(* Logix 5000 project; controller HP_SSC01hv vendor 1 type 14 code 158 rev 32.11; software revision 32.03; part 3 of 15 *)
(* tags used below, declared in another part *)
   A_C1_0218 : ALIAS FOR S_C1_FaultSafety.18;
   A_C1_0219 : ALIAS FOR S_C1_FaultSafety.19;
   A_C1_0220 : ALIAS FOR S_C1_FaultSafety.20;
   A_C1_0221 : ALIAS FOR S_C1_FaultSafety.21;
   A_C1_0222 : ALIAS FOR S_C1_FaultSafety.22;
   A_C1_0223 : ALIAS FOR S_C1_FaultSafety.23;
   A_C1_0311 : ALIAS FOR C1_FaultStandard.11;
   A_C1_0312 : ALIAS FOR C1_FaultStandard.12;
   A_C1_0313 : ALIAS FOR C1_FaultStandard.13;
   A_C1_0314 : ALIAS FOR C1_FaultStandard.14;
   A_C1_0315 : ALIAS FOR C1_FaultStandard.15;
   C1_EncoderDegree : REAL;
   C1_EncoderPositionAtHome : DINT;
   C1_ExcecutePBHoldTimer : TIMER;
   C1_FaultHomeSwitchNotFound : BOOL;
   C1_Homed : BOOL;
   C1_HomeDelay : TIMER[16];
   C1_HomeFindSwitchMAM01 : MOTION_INSTRUCTION;
   C1_HomeFindSwitchMAM02 : MOTION_INSTRUCTION;
   C1_HomeFindSwitchMAS01 : MOTION_INSTRUCTION;
   C1_HomeGetCloseToSwitchMAM01 : MOTION_INSTRUCTION;
   C1_HomeGoToOnPathMAM01 : MOTION_INSTRUCTION;
   C1_HomeMessageNumber : DINT;
   C1_HomeSensorTestMAM02 : MOTION_INSTRUCTION;
   C1_HomeSequence : DINT;
   C1_HomeSequenceAlarms : DINT;
   C1_HomeSequenceAlarmTimer : TIMER[32];
   C1_HomeSequenceInProcess : BOOL;
   C1_HomeSequenceMAH : MOTION_INSTRUCTION;
   C1_HomeSwitchFaultK7KFailedOff : BOOL;
   C1_HomeSwitchFaultK7KFailedOn : BOOL;
   C1_HomeSwitchFaultSafeFailedOff : BOOL;
   C1_HomeSwitchFaultSafeFailedOn : BOOL;
   C1_HomeTest : REAL;
   C1_IndexEnable : BOOL;
   C1_IndexEnableTOF : TIMER;
   C1_IndexMAM01 : MOTION_INSTRUCTION;
   C1_IndexMAS01 : MOTION_INSTRUCTION;
   C1_IndexMessageNumber : DINT;
   C1_IndexPermissive : BOOL;
   C1_Jog_ONS : DINT;
   C1_JogDirection : DINT;
   C1_JogEnable : BOOL;
   C1_JogEnableTOF : TIMER;
   C1_JogForwardFastSelected : BOOL;
   C1_JogForwardSlowSelected : BOOL;
   C1_JogMAJ01 : MOTION_INSTRUCTION;
   C1_JogMAJ02 : MOTION_INSTRUCTION;
   C1_JogMAS01 : MOTION_INSTRUCTION;
   C1_JogMessageNumber : DINT;
   C1_JogPermissive : BOOL;
   C1_JogReverseFastSelected : BOOL;
   C1_JogReverseSlowSelected : BOOL;
   C1_MAJAcceleration : REAL;
   C1_MAJDeceleration : REAL;
   C1_MAJSpeed : REAL;
   C1_OIT_Current : DINT;
   C1_RemoteHomeCMD : BOOL;
   C1_ServoActionStatusOnDelay : TIMER;
   C1_SetEncoderHomePosition : BOOL;
   C1HomeSensorTestMAM01 : MOTION_INSTRUCTION;
   C1HomeSequenceONS : BOOL;
   C1HomeSequenceONS2 : BOOL;
   none : BOOL;
   S_C1_EncoderPositionAtHomeSet : BOOL;
   S_C1_ExecutePB : BOOL;
   S_C1_FaultReset : BOOL;
   S_C1_HomeSafePE : ALIAS FOR C1_Safe:I.Pt04Data;
   S_C1_ModeLocal : BOOL;
   S_C1_ModeRemote : BOOL;
   S_C1_MSTOP_InputOK : BOOL;
   S_EncoderCtsFor360Deg : DINT;
(* Carousel1, continued *)

ROUTINE C130_Home   (* ladder *)
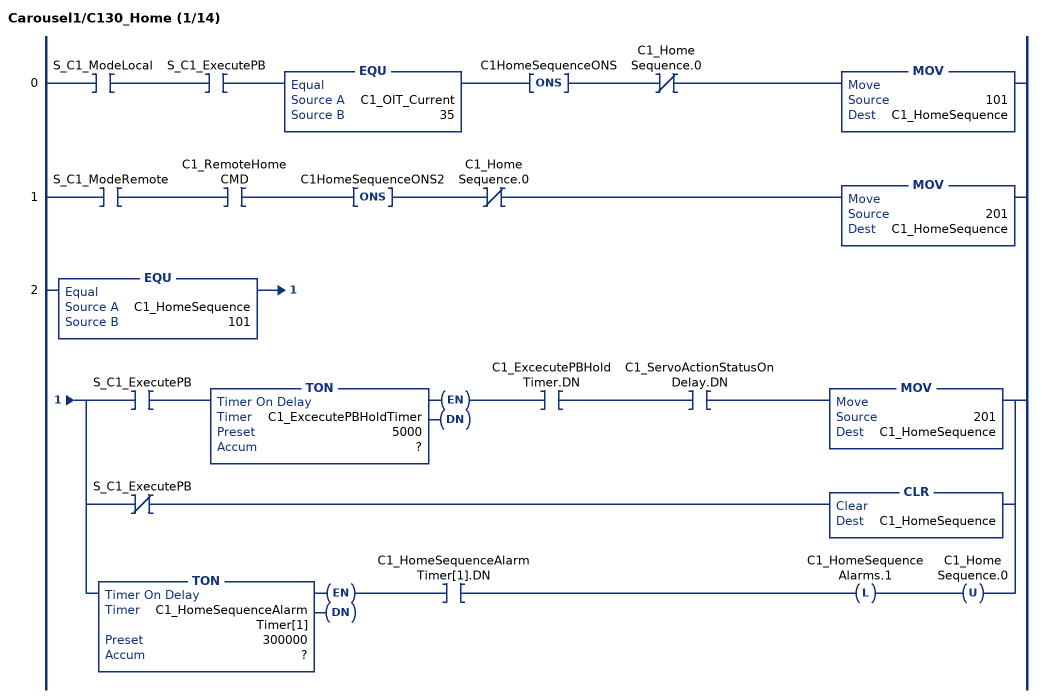
   0: XIC(S_C1_ModeLocal)XIC(S_C1_ExecutePB)EQU(C1_OIT_Current,35)ONS(C1HomeSequenceONS)XIO(C1_HomeSequence.0)MOV(101,C1_HomeSequence);
   1: XIC(S_C1_ModeRemote)XIC(C1_RemoteHomeCMD)ONS(C1HomeSequenceONS2)XIO(C1_HomeSequence.0)MOV(201,C1_HomeSequence);
   2: EQU(C1_HomeSequence,101)[XIC(S_C1_ExecutePB) TON(C1_ExcecutePBHoldTimer,?,?) XIC(C1_ExcecutePBHoldTimer.DN) XIC(C1_ServoActionStatusOnDelay.DN) MOV(201,C1_HomeSequence) ,XIO(S_C1_ExecutePB) CLR(C1_HomeSequence) ,TON(C1_HomeSequenceAlarmTimer[1],?,?) XIC(C1_HomeSequenceAlarmTimer[1].DN) OTL(C1_HomeSequenceAlarms.1) OTU(C1_HomeSequence.0) ];
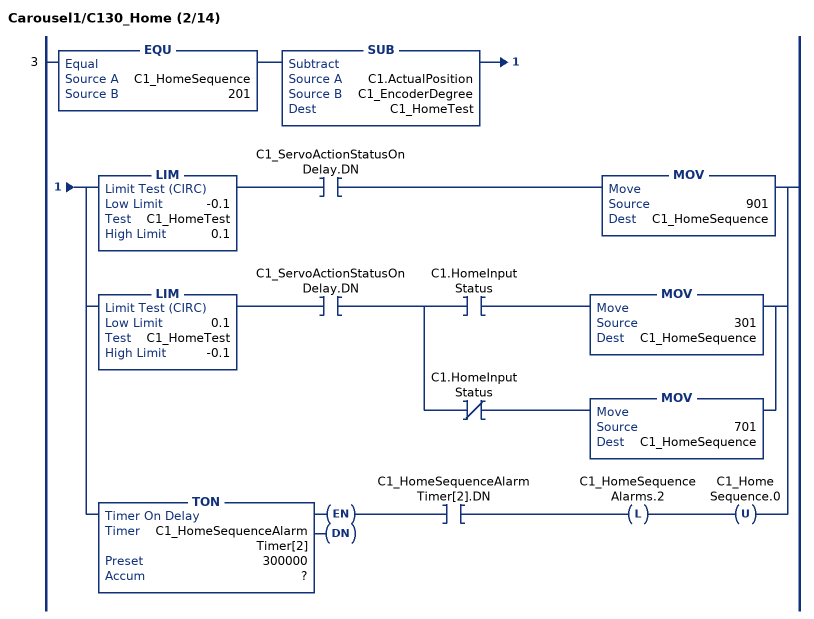
   3: EQU(C1_HomeSequence,201)SUB(C1.ActualPosition,C1_EncoderDegree,C1_HomeTest)[LIM(-0.1,C1_HomeTest,0.1) XIC(C1_ServoActionStatusOnDelay.DN) MOV(901,C1_HomeSequence) ,LIM(0.1,C1_HomeTest,-0.1) XIC(C1_ServoActionStatusOnDelay.DN) [XIC(C1.HomeInputStatus) MOV(301,C1_HomeSequence) ,XIO(C1.HomeInputStatus) MOV(701,C1_HomeSequence) ] ,TON(C1_HomeSequenceAlarmTimer[2],?,?) XIC(C1_HomeSequenceAlarmTimer[2].DN) OTL(C1_HomeSequenceAlarms.2) OTU(C1_HomeSequence.0) ];
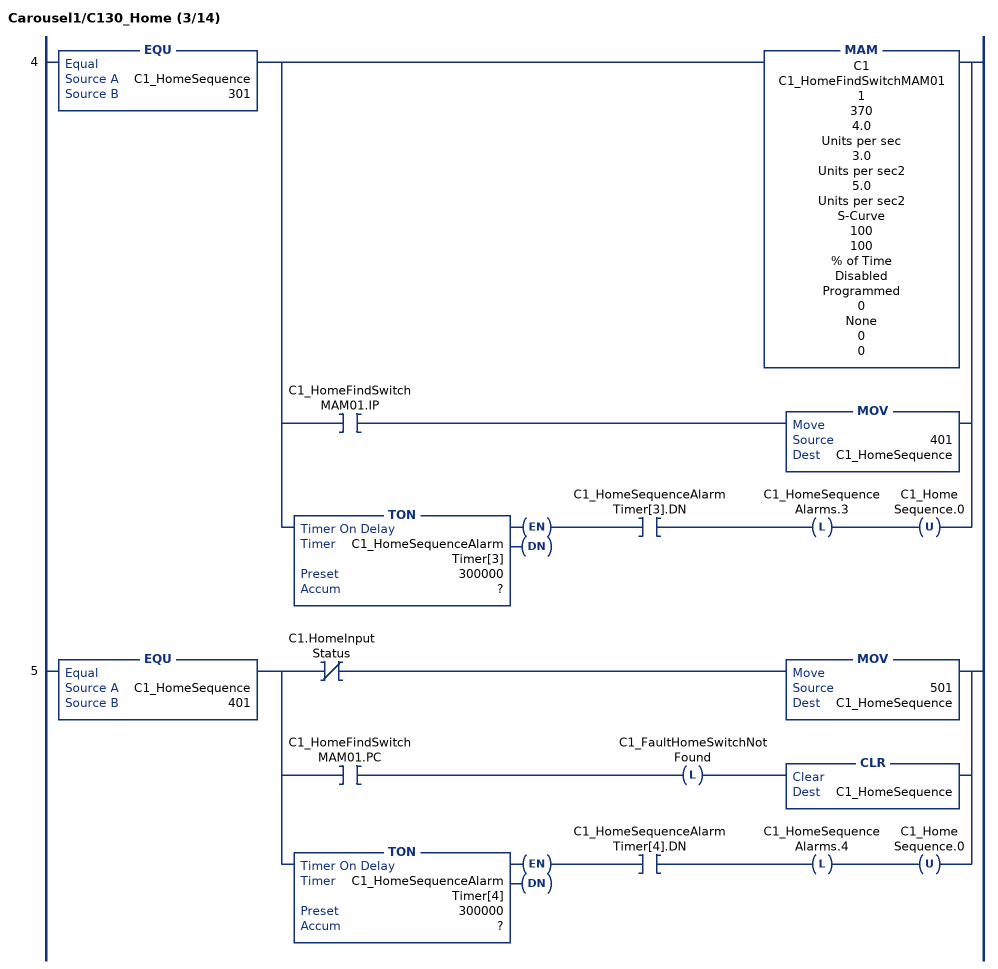
   4: EQU(C1_HomeSequence,301)[MAM(C1,C1_HomeFindSwitchMAM01,1,370,4.0,Units per sec,3.0,Units per sec2,5.0,Units per sec2,S-Curve,100,100,% of Time,Disabled,Programmed,0,None,0,0) ,XIC(C1_HomeFindSwitchMAM01.IP) MOV(401,C1_HomeSequence) ,TON(C1_HomeSequenceAlarmTimer[3],?,?) XIC(C1_HomeSequenceAlarmTimer[3].DN) OTL(C1_HomeSequenceAlarms.3) OTU(C1_HomeSequence.0) ];
   5: EQU(C1_HomeSequence,401)[XIO(C1.HomeInputStatus) MOV(501,C1_HomeSequence) ,XIC(C1_HomeFindSwitchMAM01.PC) OTL(C1_FaultHomeSwitchNotFound) CLR(C1_HomeSequence) ,TON(C1_HomeSequenceAlarmTimer[4],?,?) XIC(C1_HomeSequenceAlarmTimer[4].DN) OTL(C1_HomeSequenceAlarms.4) OTU(C1_HomeSequence.0) ];
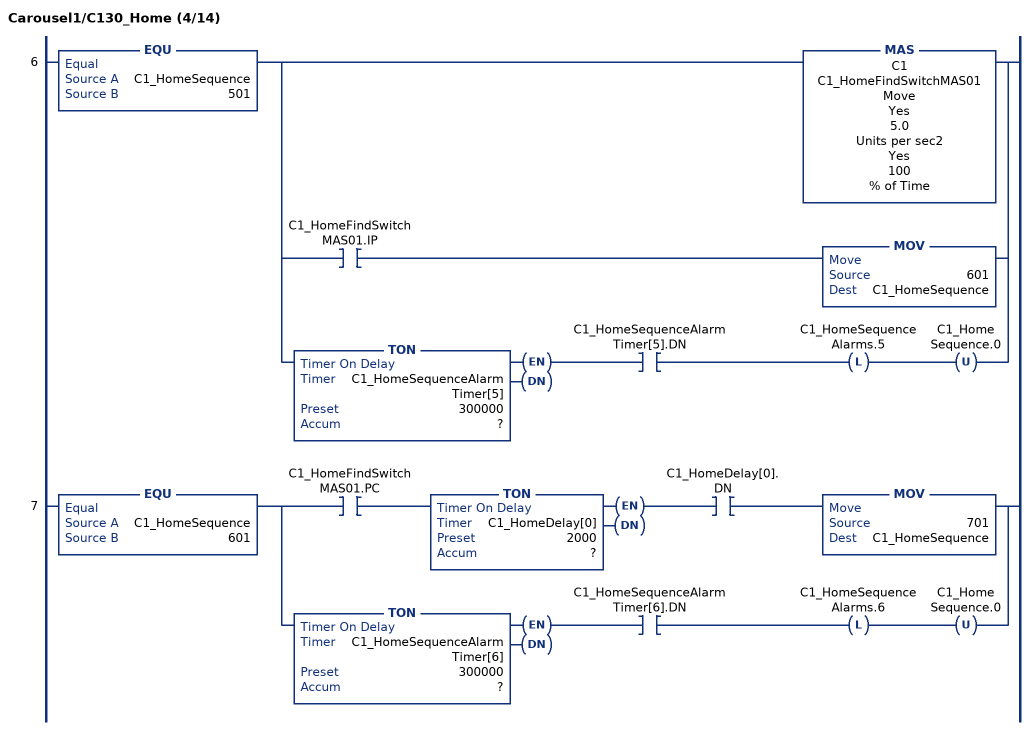
   6: EQU(C1_HomeSequence,501)[MAS(C1,C1_HomeFindSwitchMAS01,Move,Yes,5.0,Units per sec2,Yes,100,% of Time) ,XIC(C1_HomeFindSwitchMAS01.IP) MOV(601,C1_HomeSequence) ,TON(C1_HomeSequenceAlarmTimer[5],?,?) XIC(C1_HomeSequenceAlarmTimer[5].DN) OTL(C1_HomeSequenceAlarms.5) OTU(C1_HomeSequence.0) ];
   7: EQU(C1_HomeSequence,601)[XIC(C1_HomeFindSwitchMAS01.PC) TON(C1_HomeDelay[0],?,?) XIC(C1_HomeDelay[0].DN) MOV(701,C1_HomeSequence) ,TON(C1_HomeSequenceAlarmTimer[6],?,?) XIC(C1_HomeSequenceAlarmTimer[6].DN) OTL(C1_HomeSequenceAlarms.6) OTU(C1_HomeSequence.0) ];
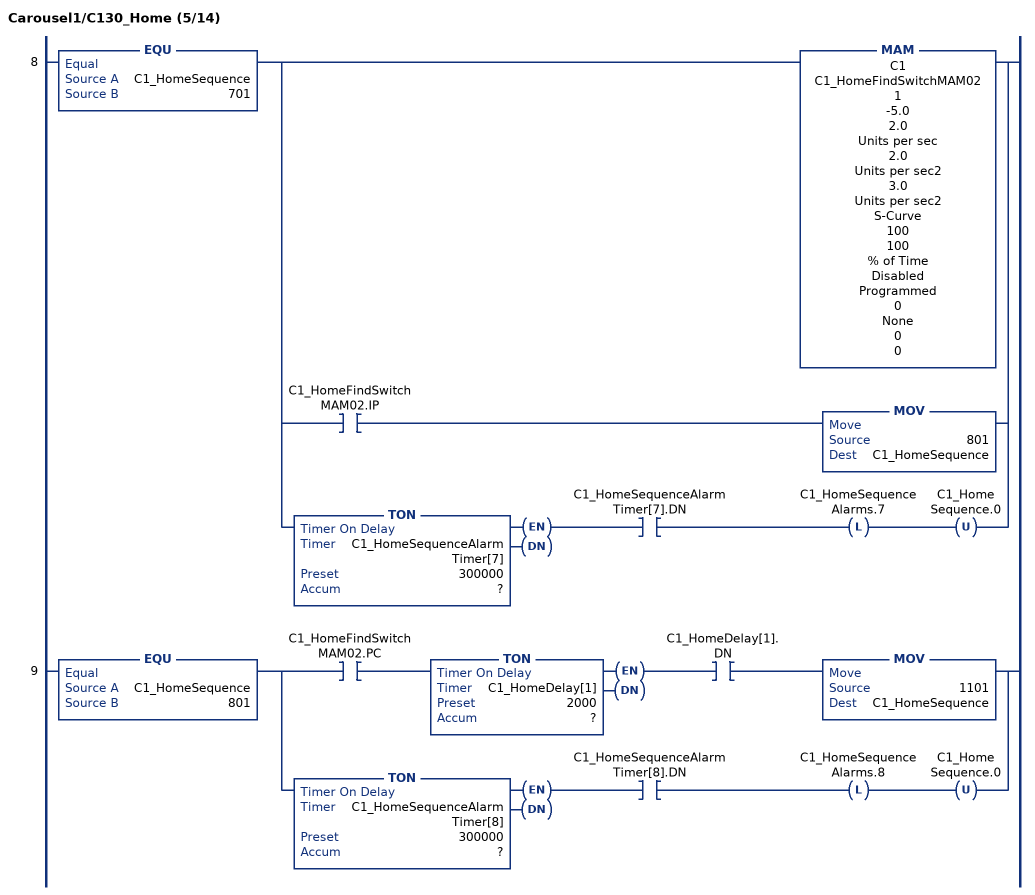
   8: EQU(C1_HomeSequence,701)[MAM(C1,C1_HomeFindSwitchMAM02,1,-5.0,2.0,Units per sec,2.0,Units per sec2,3.0,Units per sec2,S-Curve,100,100,% of Time,Disabled,Programmed,0,None,0,0) ,XIC(C1_HomeFindSwitchMAM02.IP) MOV(801,C1_HomeSequence) ,TON(C1_HomeSequenceAlarmTimer[7],?,?) XIC(C1_HomeSequenceAlarmTimer[7].DN) OTL(C1_HomeSequenceAlarms.7) OTU(C1_HomeSequence.0) ];
   9: EQU(C1_HomeSequence,801)[XIC(C1_HomeFindSwitchMAM02.PC) TON(C1_HomeDelay[1],?,?) XIC(C1_HomeDelay[1].DN) MOV(1101,C1_HomeSequence) ,TON(C1_HomeSequenceAlarmTimer[8],?,?) XIC(C1_HomeSequenceAlarmTimer[8].DN) OTL(C1_HomeSequenceAlarms.8) OTU(C1_HomeSequence.0) ];
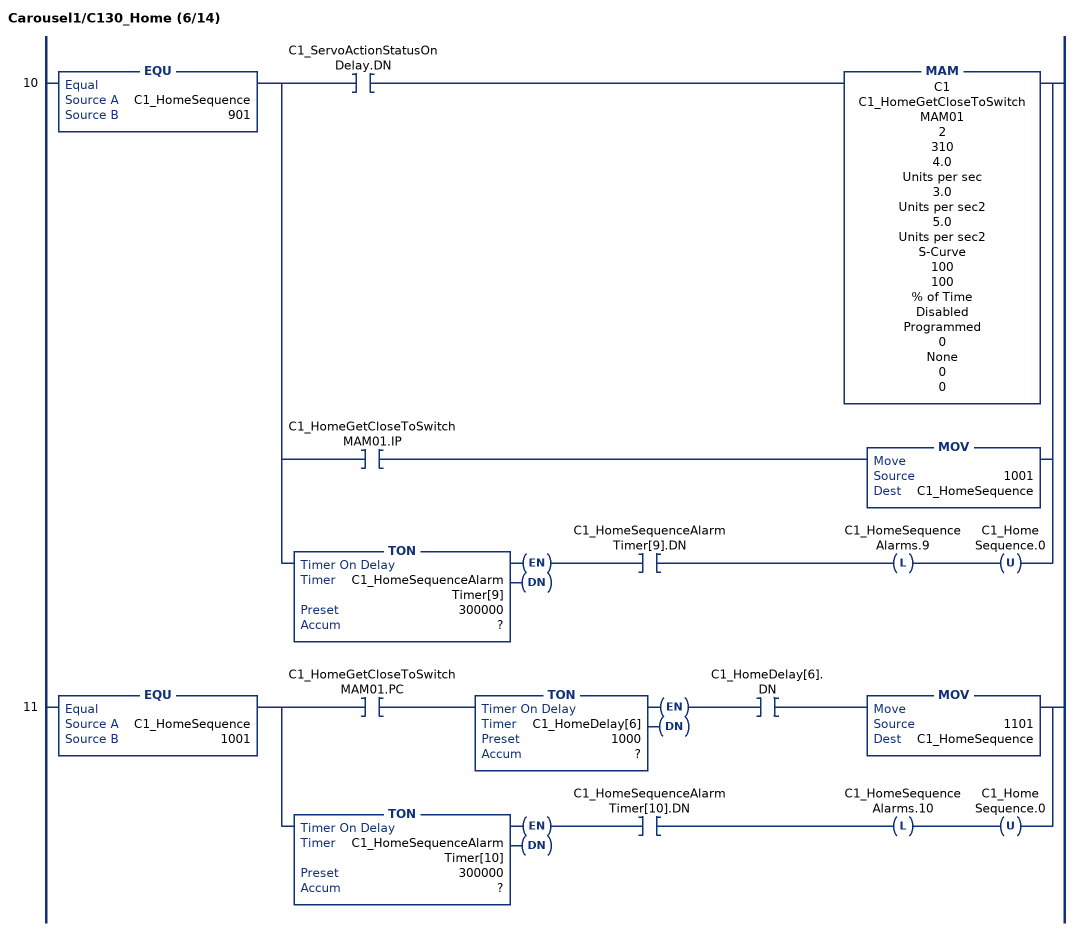
   10: EQU(C1_HomeSequence,901)[XIC(C1_ServoActionStatusOnDelay.DN) MAM(C1,C1_HomeGetCloseToSwitchMAM01,2,310,4.0,Units per sec,3.0,Units per sec2,5.0,Units per sec2,S-Curve,100,100,% of Time,Disabled,Programmed,0,None,0,0) ,XIC(C1_HomeGetCloseToSwitchMAM01.IP) MOV(1001,C1_HomeSequence) ,TON(C1_HomeSequenceAlarmTimer[9],?,?) XIC(C1_HomeSequenceAlarmTimer[9].DN) OTL(C1_HomeSequenceAlarms.9) OTU(C1_HomeSequence.0) ];
   11: EQU(C1_HomeSequence,1001)[XIC(C1_HomeGetCloseToSwitchMAM01.PC) TON(C1_HomeDelay[6],?,?) XIC(C1_HomeDelay[6].DN) MOV(1101,C1_HomeSequence) ,TON(C1_HomeSequenceAlarmTimer[10],?,?) XIC(C1_HomeSequenceAlarmTimer[10].DN) OTL(C1_HomeSequenceAlarms.10) OTU(C1_HomeSequence.0) ];
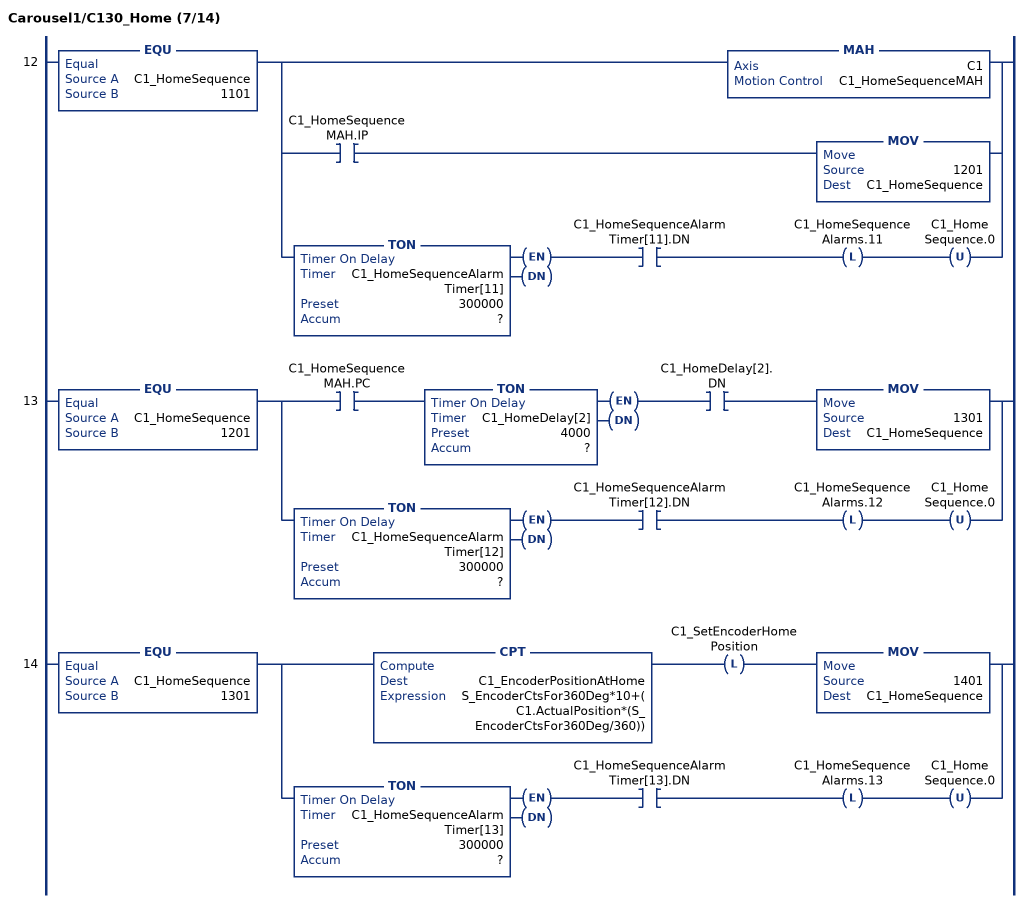
   12: EQU(C1_HomeSequence,1101)[MAH(C1,C1_HomeSequenceMAH) ,XIC(C1_HomeSequenceMAH.IP) MOV(1201,C1_HomeSequence) ,TON(C1_HomeSequenceAlarmTimer[11],?,?) XIC(C1_HomeSequenceAlarmTimer[11].DN) OTL(C1_HomeSequenceAlarms.11) OTU(C1_HomeSequence.0) ];
   13: EQU(C1_HomeSequence,1201)[XIC(C1_HomeSequenceMAH.PC) TON(C1_HomeDelay[2],?,?) XIC(C1_HomeDelay[2].DN) MOV(1301,C1_HomeSequence) ,TON(C1_HomeSequenceAlarmTimer[12],?,?) XIC(C1_HomeSequenceAlarmTimer[12].DN) OTL(C1_HomeSequenceAlarms.12) OTU(C1_HomeSequence.0) ];
   14: EQU(C1_HomeSequence,1301)[CPT(C1_EncoderPositionAtHome,S_EncoderCtsFor360Deg*10+(C1.ActualPosition*(S_EncoderCtsFor360Deg/360))) OTL(C1_SetEncoderHomePosition) MOV(1401,C1_HomeSequence) ,TON(C1_HomeSequenceAlarmTimer[13],?,?) XIC(C1_HomeSequenceAlarmTimer[13].DN) OTL(C1_HomeSequenceAlarms.13) OTU(C1_HomeSequence.0) ];
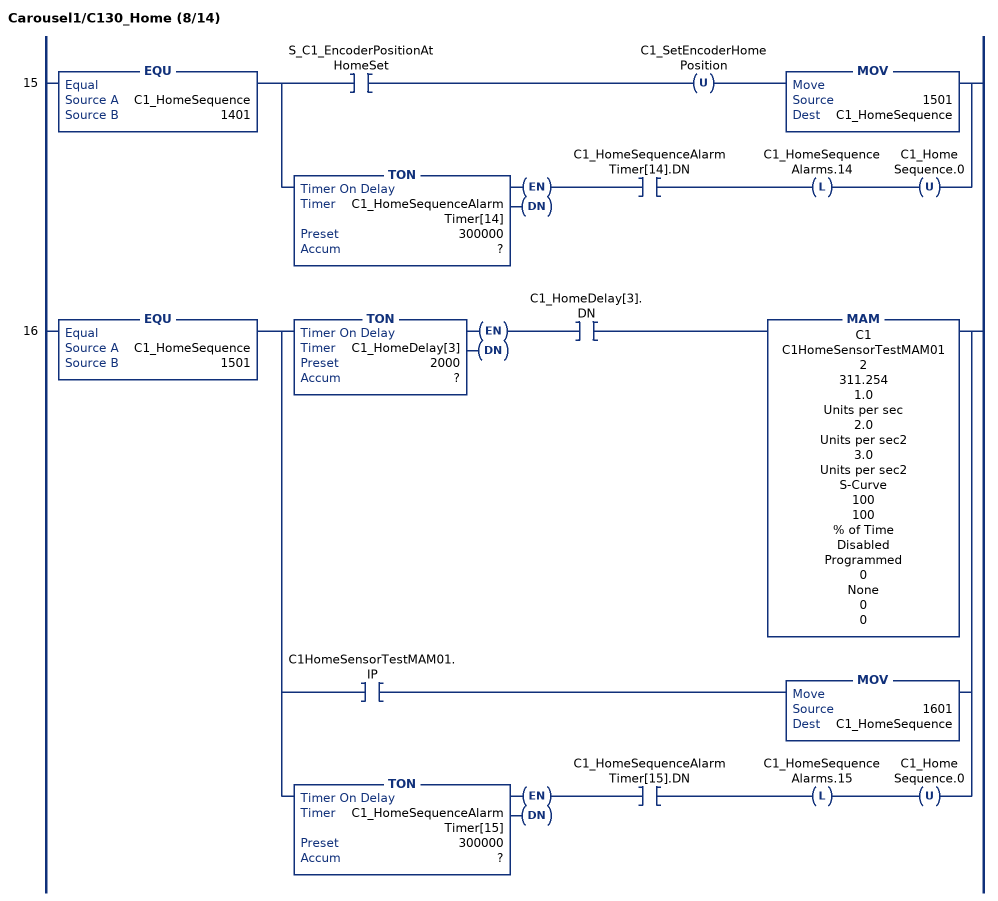
   15: EQU(C1_HomeSequence,1401)[XIC(S_C1_EncoderPositionAtHomeSet) OTU(C1_SetEncoderHomePosition) MOV(1501,C1_HomeSequence) ,TON(C1_HomeSequenceAlarmTimer[14],?,?) XIC(C1_HomeSequenceAlarmTimer[14].DN) OTL(C1_HomeSequenceAlarms.14) OTU(C1_HomeSequence.0) ];
   16: EQU(C1_HomeSequence,1501)[TON(C1_HomeDelay[3],?,?) XIC(C1_HomeDelay[3].DN) MAM(C1,C1HomeSensorTestMAM01,2,311.254,1.0,Units per sec,2.0,Units per sec2,3.0,Units per sec2,S-Curve,100,100,% of Time,Disabled,Programmed,0,None,0,0) ,XIC(C1HomeSensorTestMAM01.IP) MOV(1601,C1_HomeSequence) ,TON(C1_HomeSequenceAlarmTimer[15],?,?) XIC(C1_HomeSequenceAlarmTimer[15].DN) OTL(C1_HomeSequenceAlarms.15) OTU(C1_HomeSequence.0) ];
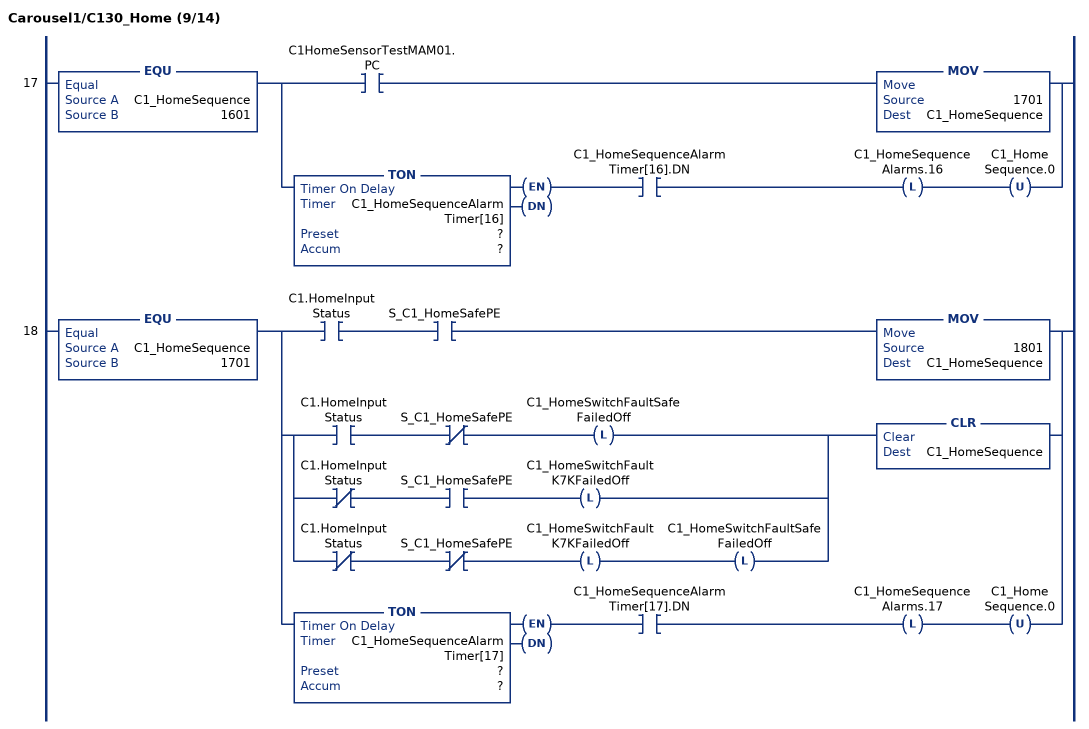
   17: EQU(C1_HomeSequence,1601)[XIC(C1HomeSensorTestMAM01.PC) MOV(1701,C1_HomeSequence) ,TON(C1_HomeSequenceAlarmTimer[16],?,?) XIC(C1_HomeSequenceAlarmTimer[16].DN) OTL(C1_HomeSequenceAlarms.16) OTU(C1_HomeSequence.0) ];
   18: EQU(C1_HomeSequence,1701)[XIC(C1.HomeInputStatus) XIC(S_C1_HomeSafePE) MOV(1801,C1_HomeSequence) ,[XIC(C1.HomeInputStatus) XIO(S_C1_HomeSafePE) OTL(C1_HomeSwitchFaultSafeFailedOff) ,XIO(C1.HomeInputStatus) XIC(S_C1_HomeSafePE) OTL(C1_HomeSwitchFaultK7KFailedOff) ,XIO(C1.HomeInputStatus) XIO(S_C1_HomeSafePE) OTL(C1_HomeSwitchFaultK7KFailedOff) OTL(C1_HomeSwitchFaultSafeFailedOff) ] CLR(C1_HomeSequence) ,TON(C1_HomeSequenceAlarmTimer[17],?,?) XIC(C1_HomeSequenceAlarmTimer[17].DN) OTL(C1_HomeSequenceAlarms.17) OTU(C1_HomeSequence.0) ];
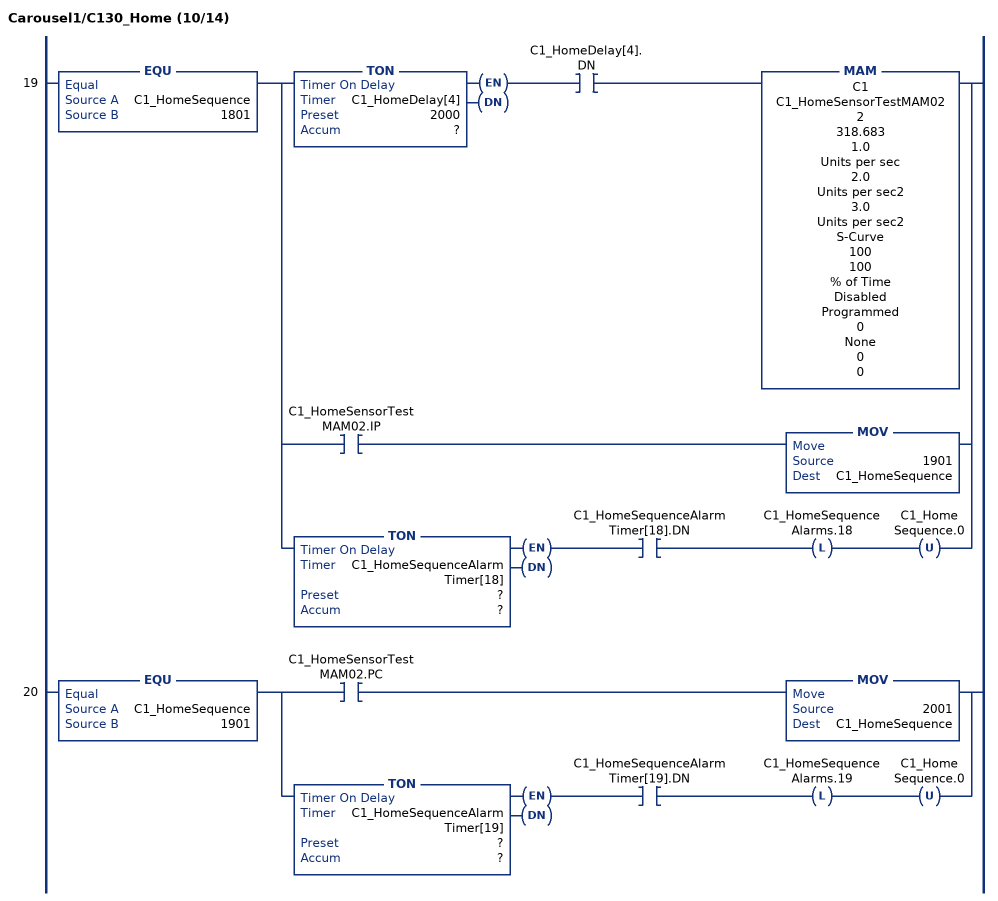
   19: EQU(C1_HomeSequence,1801)[TON(C1_HomeDelay[4],?,?) XIC(C1_HomeDelay[4].DN) MAM(C1,C1_HomeSensorTestMAM02,2,318.683,1.0,Units per sec,2.0,Units per sec2,3.0,Units per sec2,S-Curve,100,100,% of Time,Disabled,Programmed,0,None,0,0) ,XIC(C1_HomeSensorTestMAM02.IP) MOV(1901,C1_HomeSequence) ,TON(C1_HomeSequenceAlarmTimer[18],?,?) XIC(C1_HomeSequenceAlarmTimer[18].DN) OTL(C1_HomeSequenceAlarms.18) OTU(C1_HomeSequence.0) ];
   20: EQU(C1_HomeSequence,1901)[XIC(C1_HomeSensorTestMAM02.PC) MOV(2001,C1_HomeSequence) ,TON(C1_HomeSequenceAlarmTimer[19],?,?) XIC(C1_HomeSequenceAlarmTimer[19].DN) OTL(C1_HomeSequenceAlarms.19) OTU(C1_HomeSequence.0) ];
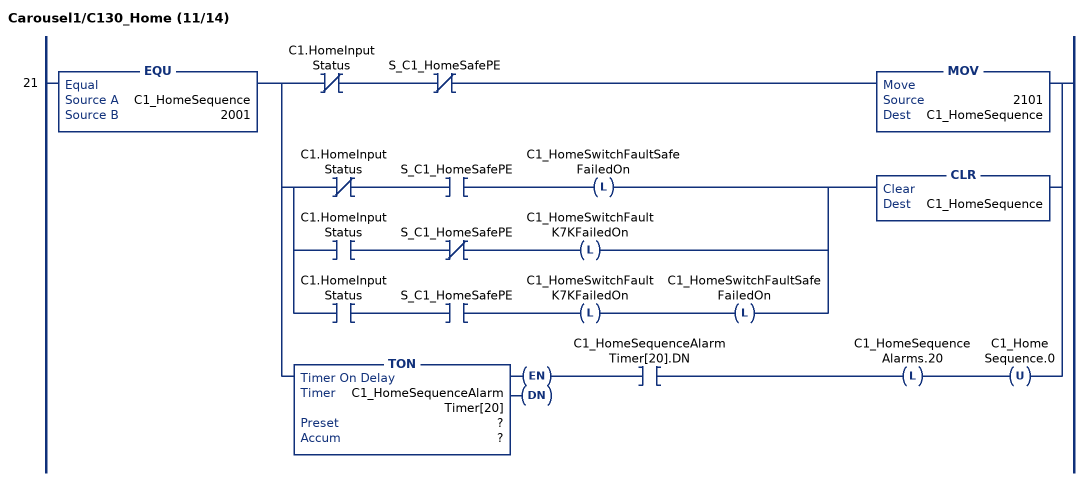
   21: EQU(C1_HomeSequence,2001)[XIO(C1.HomeInputStatus) XIO(S_C1_HomeSafePE) MOV(2101,C1_HomeSequence) ,[XIO(C1.HomeInputStatus) XIC(S_C1_HomeSafePE) OTL(C1_HomeSwitchFaultSafeFailedOn) ,XIC(C1.HomeInputStatus) XIO(S_C1_HomeSafePE) OTL(C1_HomeSwitchFaultK7KFailedOn) ,XIC(C1.HomeInputStatus) XIC(S_C1_HomeSafePE) OTL(C1_HomeSwitchFaultK7KFailedOn) OTL(C1_HomeSwitchFaultSafeFailedOn) ] CLR(C1_HomeSequence) ,TON(C1_HomeSequenceAlarmTimer[20],?,?) XIC(C1_HomeSequenceAlarmTimer[20].DN) OTL(C1_HomeSequenceAlarms.20) OTU(C1_HomeSequence.0) ];
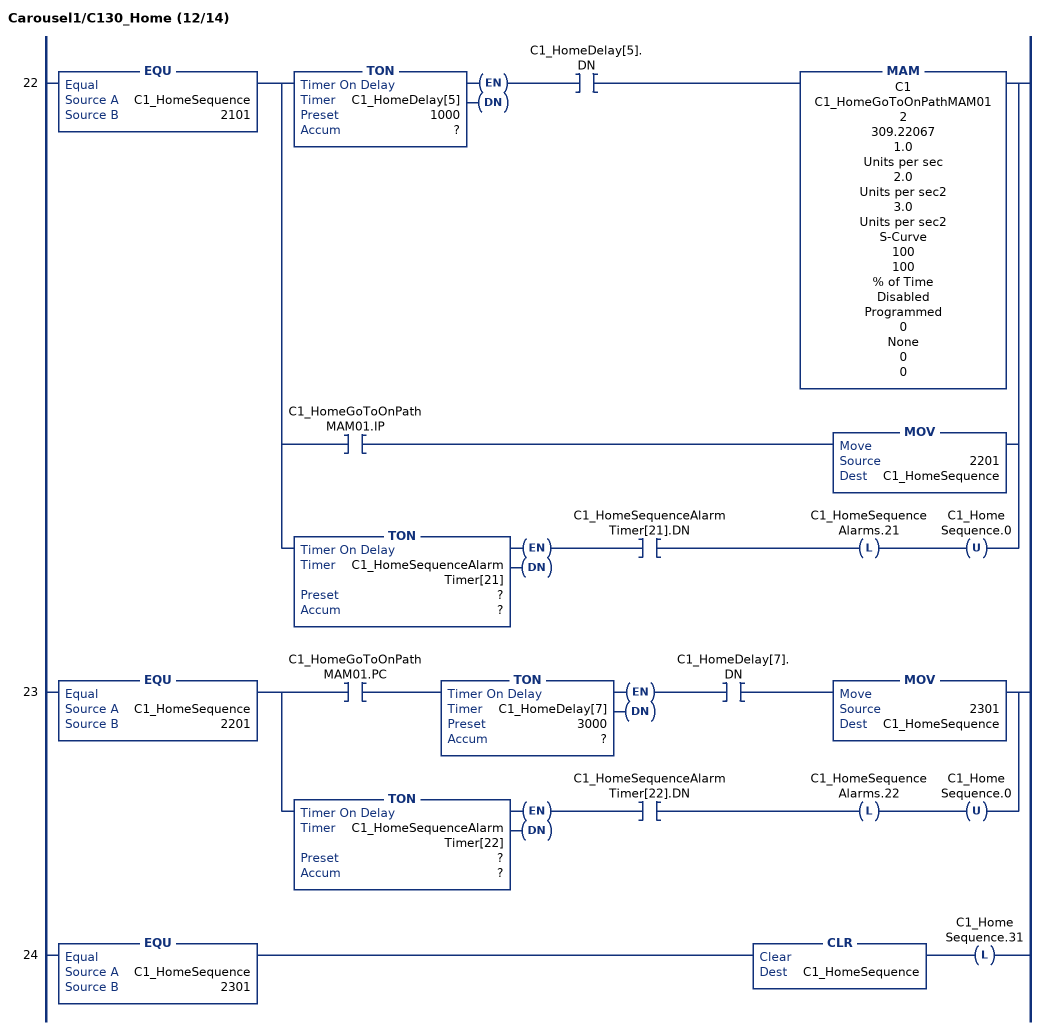
   22: EQU(C1_HomeSequence,2101)[TON(C1_HomeDelay[5],?,?) XIC(C1_HomeDelay[5].DN) MAM(C1,C1_HomeGoToOnPathMAM01,2,309.22067,1.0,Units per sec,2.0,Units per sec2,3.0,Units per sec2,S-Curve,100,100,% of Time,Disabled,Programmed,0,None,0,0) ,XIC(C1_HomeGoToOnPathMAM01.IP) MOV(2201,C1_HomeSequence) ,TON(C1_HomeSequenceAlarmTimer[21],?,?) XIC(C1_HomeSequenceAlarmTimer[21].DN) OTL(C1_HomeSequenceAlarms.21) OTU(C1_HomeSequence.0) ];
   23: EQU(C1_HomeSequence,2201)[XIC(C1_HomeGoToOnPathMAM01.PC) TON(C1_HomeDelay[7],?,?) XIC(C1_HomeDelay[7].DN) MOV(2301,C1_HomeSequence) ,TON(C1_HomeSequenceAlarmTimer[22],?,?) XIC(C1_HomeSequenceAlarmTimer[22].DN) OTL(C1_HomeSequenceAlarms.22) OTU(C1_HomeSequence.0) ];
   24: EQU(C1_HomeSequence,2301)CLR(C1_HomeSequence)OTL(C1_HomeSequence.31);
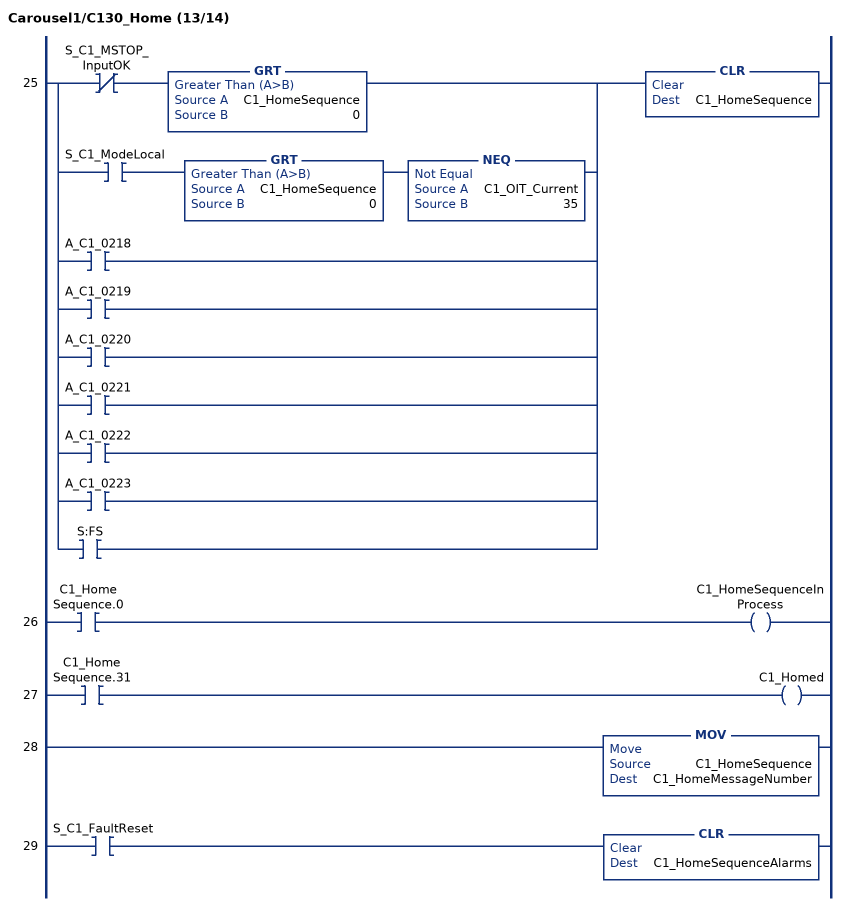
   25: [XIO(S_C1_MSTOP_InputOK) GRT(C1_HomeSequence,0) ,XIC(S_C1_ModeLocal) GRT(C1_HomeSequence,0) NEQ(C1_OIT_Current,35) ,XIC(A_C1_0218) ,XIC(A_C1_0219) ,XIC(A_C1_0220) ,XIC(A_C1_0221) ,XIC(A_C1_0222) ,XIC(A_C1_0223) ,XIC(S:FS) ]CLR(C1_HomeSequence);
   26: XIC(C1_HomeSequence.0)OTE(C1_HomeSequenceInProcess);
   27: XIC(C1_HomeSequence.31)OTE(C1_Homed);
   28: MOV(C1_HomeSequence,C1_HomeMessageNumber);
   29: XIC(S_C1_FaultReset)CLR(C1_HomeSequenceAlarms);
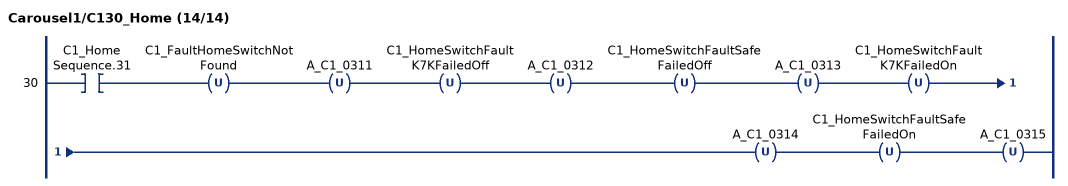
   30: XIC(C1_HomeSequence.31)OTU(C1_FaultHomeSwitchNotFound)OTU(A_C1_0311)OTU(C1_HomeSwitchFaultK7KFailedOff)OTU(A_C1_0312)OTU(C1_HomeSwitchFaultSafeFailedOff)OTU(A_C1_0313)OTU(C1_HomeSwitchFaultK7KFailedOn)OTU(A_C1_0314)OTU(C1_HomeSwitchFaultSafeFailedOn)OTU(A_C1_0315);
END_ROUTINE

ROUTINE C135_Index   (* ladder *)
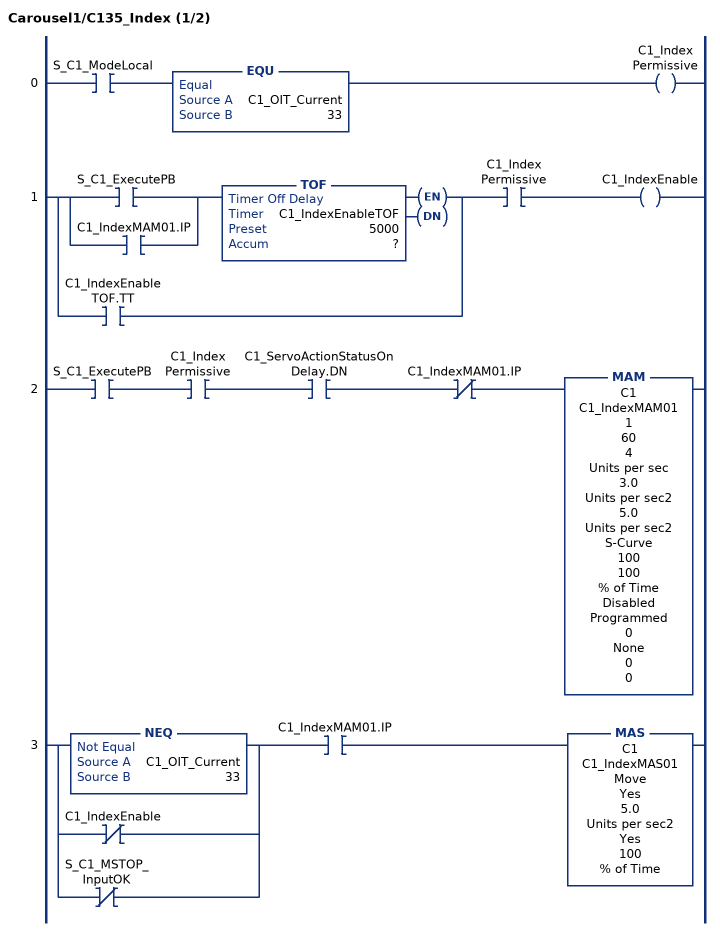
   0: XIC(S_C1_ModeLocal)EQU(C1_OIT_Current,33)OTE(C1_IndexPermissive);
   1: [[XIC(S_C1_ExecutePB) ,XIC(C1_IndexMAM01.IP) ] TOF(C1_IndexEnableTOF,?,?) ,XIC(C1_IndexEnableTOF.TT) ]XIC(C1_IndexPermissive)OTE(C1_IndexEnable);
   2: XIC(S_C1_ExecutePB)XIC(C1_IndexPermissive)XIC(C1_ServoActionStatusOnDelay.DN)XIO(C1_IndexMAM01.IP)MAM(C1,C1_IndexMAM01,1,60,4,Units per sec,3.0,Units per sec2,5.0,Units per sec2,S-Curve,100,100,% of Time,Disabled,Programmed,0,None,0,0);
   3: [NEQ(C1_OIT_Current,33) ,XIO(C1_IndexEnable) ,XIO(S_C1_MSTOP_InputOK) ]XIC(C1_IndexMAM01.IP)MAS(C1,C1_IndexMAS01,Move,Yes,5.0,Units per sec2,Yes,100,% of Time);
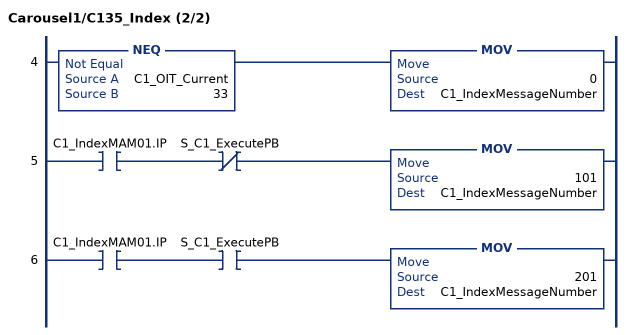
   4: NEQ(C1_OIT_Current,33)MOV(0,C1_IndexMessageNumber);
   5: XIC(C1_IndexMAM01.IP)XIO(S_C1_ExecutePB)MOV(101,C1_IndexMessageNumber);
   6: XIC(C1_IndexMAM01.IP)XIC(S_C1_ExecutePB)MOV(201,C1_IndexMessageNumber);
END_ROUTINE

ROUTINE C140_Jog   (* ladder *)
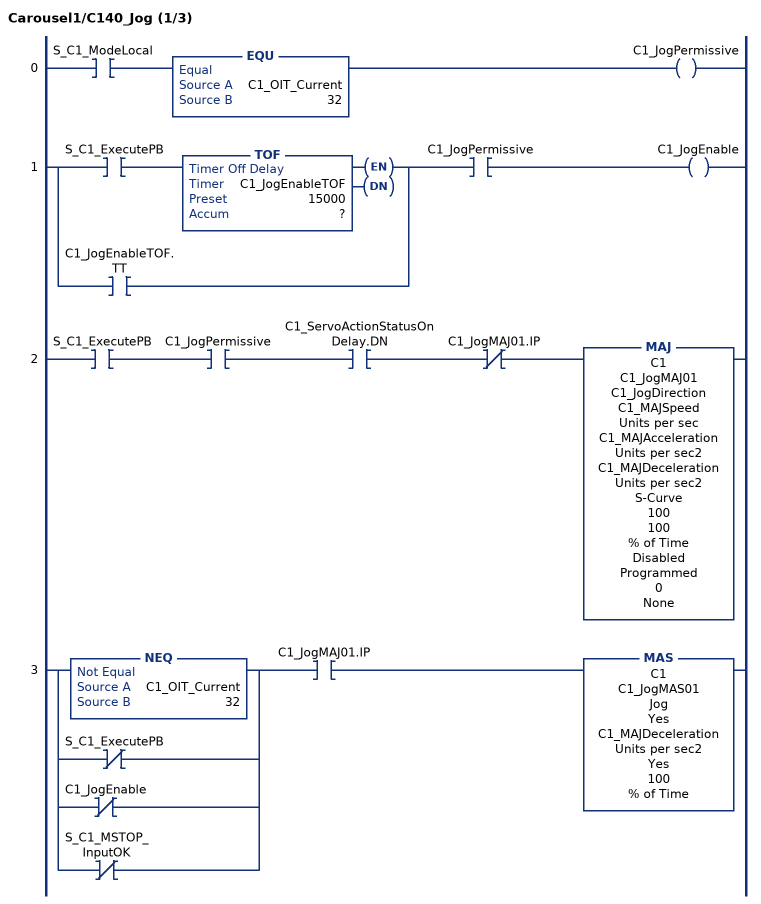
   0: XIC(S_C1_ModeLocal)EQU(C1_OIT_Current,32)OTE(C1_JogPermissive);
   1: [XIC(S_C1_ExecutePB) TOF(C1_JogEnableTOF,?,?) ,XIC(C1_JogEnableTOF.TT) ]XIC(C1_JogPermissive)OTE(C1_JogEnable);
   2: XIC(S_C1_ExecutePB)XIC(C1_JogPermissive)XIC(C1_ServoActionStatusOnDelay.DN)XIO(C1_JogMAJ01.IP)MAJ(C1,C1_JogMAJ01,C1_JogDirection,C1_MAJSpeed,Units per sec,C1_MAJAcceleration,Units per sec2,C1_MAJDeceleration,Units per sec2,S-Curve,100,100,% of Time,Disabled,Programmed,0,None);
   3: [NEQ(C1_OIT_Current,32) ,XIO(S_C1_ExecutePB) ,XIO(C1_JogEnable) ,XIO(S_C1_MSTOP_InputOK) ]XIC(C1_JogMAJ01.IP)MAS(C1,C1_JogMAS01,Jog,Yes,C1_MAJDeceleration,Units per sec2,Yes,100,% of Time);
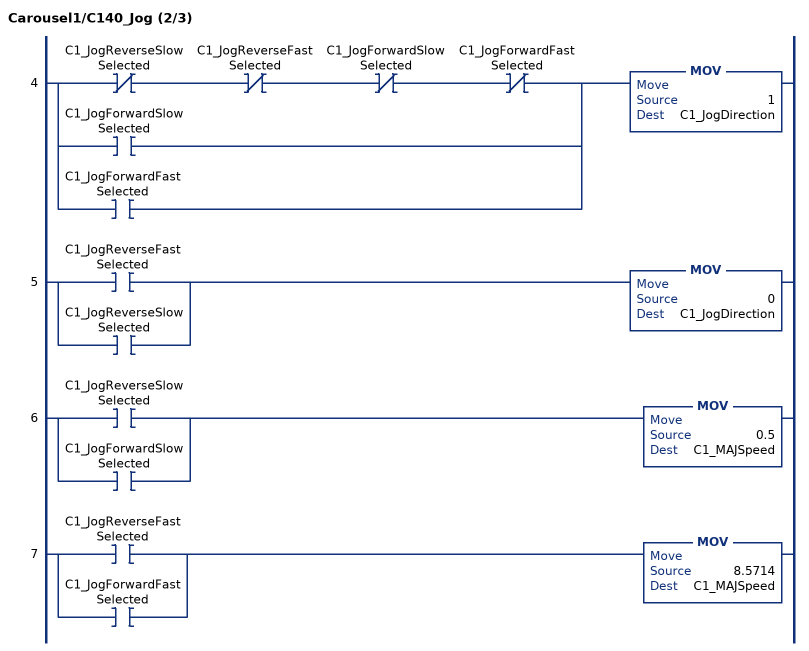
   4: [XIO(C1_JogReverseSlowSelected) XIO(C1_JogReverseFastSelected) XIO(C1_JogForwardSlowSelected) XIO(C1_JogForwardFastSelected) ,XIC(C1_JogForwardSlowSelected) ,XIC(C1_JogForwardFastSelected) ]MOV(1,C1_JogDirection);
   5: [XIC(C1_JogReverseFastSelected) ,XIC(C1_JogReverseSlowSelected) ]MOV(0,C1_JogDirection);
   6: [XIC(C1_JogReverseSlowSelected) ,XIC(C1_JogForwardSlowSelected) ]MOV(0.5,C1_MAJSpeed);
   7: [XIC(C1_JogReverseFastSelected) ,XIC(C1_JogForwardFastSelected) ]MOV(8.5714,C1_MAJSpeed);
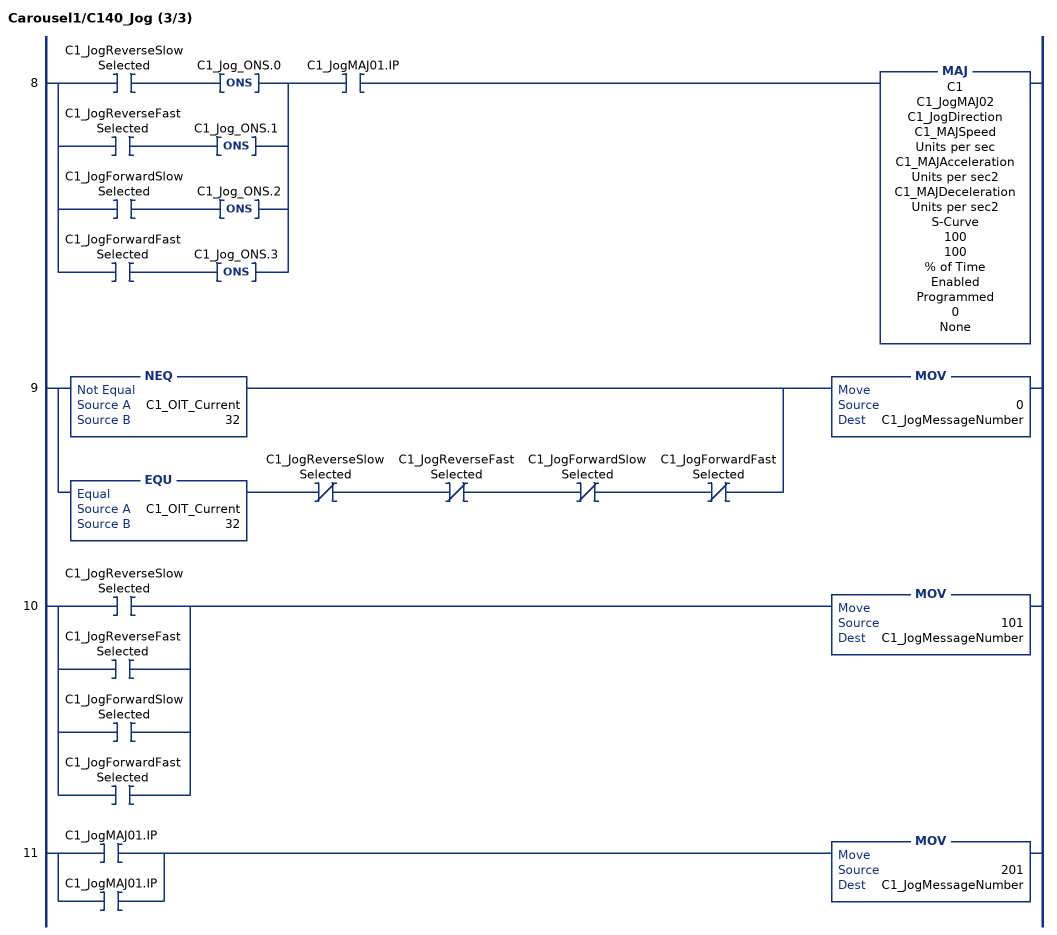
   8: [XIC(C1_JogReverseSlowSelected) ONS(C1_Jog_ONS.0) ,XIC(C1_JogReverseFastSelected) ONS(C1_Jog_ONS.1) ,XIC(C1_JogForwardSlowSelected) ONS(C1_Jog_ONS.2) ,XIC(C1_JogForwardFastSelected) ONS(C1_Jog_ONS.3) ]XIC(C1_JogMAJ01.IP)MAJ(C1,C1_JogMAJ02,C1_JogDirection,C1_MAJSpeed,Units per sec,C1_MAJAcceleration,Units per sec2,C1_MAJDeceleration,Units per sec2,S-Curve,100,100,% of Time,Enabled,Programmed,0,None);
   9: [NEQ(C1_OIT_Current,32) ,EQU(C1_OIT_Current,32) XIO(C1_JogReverseSlowSelected) XIO(C1_JogReverseFastSelected) XIO(C1_JogForwardSlowSelected) XIO(C1_JogForwardFastSelected) ]MOV(0,C1_JogMessageNumber);
   10: [XIC(C1_JogReverseSlowSelected) ,XIC(C1_JogReverseFastSelected) ,XIC(C1_JogForwardSlowSelected) ,XIC(C1_JogForwardFastSelected) ]MOV(101,C1_JogMessageNumber);
   11: [XIC(C1_JogMAJ01.IP) ,XIC(C1_JogMAJ01.IP) ]MOV(201,C1_JogMessageNumber);
END_ROUTINE
